INTERFACE I_XP_Track_PLC EXTENDS I_CH_Object

{attribute 'monitoring':='call'}
PROPERTY CtsMoversOnTrack : UINT
GET
END_GET
END_PROPERTY

{attribute 'monitoring':='call'}
PROPERTY Feedback : I_XP_Feedback
GET
END_GET
END_PROPERTY

{attribute 'monitoring':='call'}
//[mm]
PROPERTY Length : LREAL
GET
END_GET
END_PROPERTY

{attribute 'monitoring':='call'}
PROPERTY Mapped : BOOL //Project is mapped to MC (McToPlc and PlcToMc)
GET
END_GET
END_PROPERTY

{attribute 'monitoring':='call'}
//Unique object ID
PROPERTY OID : OTCID
GET
END_GET
END_PROPERTY

{attribute 'monitoring':='call'}
PROPERTY PlanarTrack : REFERENCE TO MC_PlanarTrack
GET
END_GET
END_PROPERTY

(* Returns the first station on current track who has exact thsi position or is ahead
	If no station on this track, result is maybe on another track*)
METHOD StationAhedPosition : I_XP_Station
VAR_INPUT
	fPosOnTrack : LREAL;//[mm]	
END_VAR
END_METHOD

{attribute 'monitoring':='call'}
//List of interfaces to stations on this track
PROPERTY StationsOnTrack : I_CH_List
GET
END_GET
END_PROPERTY

{attribute 'monitoring':='call'}
//List of interfaces from other tracks
PROPERTY TracksAhead : I_CH_List
GET
END_GET
END_PROPERTY

{attribute 'monitoring':='call'}
//List of interfaces from other tracks
PROPERTY TracksBehinde : I_CH_List
GET
END_GET
END_PROPERTY

{attribute 'monitoring':='call'}
PROPERTY TracksEndAtThis : REFERENCE TO  ARRAY[0..(XPlanarParameterlist.N_MAX_STATIONS_AHEAD_OR_BEHIND-1)] OF I_XP_Track
GET
END_GET
END_PROPERTY

{attribute 'monitoring':='call'}
PROPERTY TracksStartFromThis : REFERENCE TO ARRAY[0..(XPlanarParameterlist.N_MAX_STATIONS_AHEAD_OR_BEHIND-1)] OF I_XP_Track
GET
END_GET
END_PROPERTY

END_INTERFACE

(* stored: Version 1.1.0.1, ProductVersion 3.1.4024.12
   Itf I_XP_Track_PLC: Id {e6e7f968-03d3-4a49-a729-42c6442c0da9}
   Property CtsMoversOnTrack: Id {a3257dbe-6eca-46f1-99cd-8564a818db88}
   Get Get: Id {3e3d2acb-3129-4e2a-b86f-7221798788aa}
   Property Feedback: Id {910900ca-e0cf-474a-b5ef-e85942e7d249}
   Get Get: Id {091b0e68-ebe4-4864-9ab6-f2038b55fb01}
   Property Length: Id {0d6552b5-faf4-4152-b9d7-fe806ca06267}
   Get Get: Id {dbe2f754-111a-4078-97a8-d4db148490e4}
   Property Mapped: Id {e540c848-2ed1-4a70-b4a2-a9cc9a04bc0a}
   Get Get: Id {27a82caa-3fe8-40aa-b250-d2d2e7494e5f}
   Property OID: Id {bd1cf5af-57a1-4927-b6f2-46edb4bf8d4c}
   Get Get: Id {442d39cf-4546-4a1a-a631-6d7be7b51430}
   Property PlanarTrack: Id {2655453e-dca2-4400-bf0b-067a2294a8f6}
   Get Get: Id {3cfbf816-5585-4cce-adb5-63e4897036bd}
   Method StationAhedPosition: Id {66046894-762c-43ad-932b-a335bdf7d057}
   Property StationsOnTrack: Id {bab9c82e-80cb-4b84-a9a8-d947fb34b427}
   Get Get: Id {fbccfe6e-bcfc-4280-834d-3732a1fcf525}
   Property TracksAhead: Id {fdb2da1a-9d03-4c17-89f5-8063a4fe9283}
   Get Get: Id {bdaf5fdc-2ae4-451c-ac6e-86f33fecc61c}
   Property TracksBehinde: Id {471485d7-74d5-464d-a7c9-64cb6cf6358c}
   Get Get: Id {c40f8818-c15e-4b1f-8a96-6cf955be010a}
   Property TracksEndAtThis: Id {b922b958-ca67-4f7e-9d79-21b272c1edc2}
   Get Get: Id {31b1c373-e3e2-4292-aa47-a31504a24fd8}
   Property TracksStartFromThis: Id {d11fa298-cafb-4258-842b-11a45220d8de}
   Get Get: Id {bd47bc51-5d4a-4d12-a9ad-c780a8623c18} *)
